TYPE Safety_Ctx :
STRUCT
	nState			: USINT;
	iSafetyEvent	: I_Emit;
END_STRUCT
END_TYPE

(* stored: Version 1.1.0.1
   DUT Safety_Ctx: Id {40f90be4-0b9e-4b8e-9d9b-78b410336993} *)
